(* Logix 5000 project; controller cal1632 1756-L62 rev 16.20; software revision 16.05; part 54 of 57 *)
(* tags used below, declared in another part *)
   FAULT : BOOL;
   p01_param_tension_deviation : REAL;
   p01r09_pb_global_reset : BOOL;
   p01r13_state : DINT;
   p25_ao_selected_speed : REAL;
   p29_ai_wa_rpm : REAL;
   p29_ai_wb_rpm : REAL;
   p29_ai_wdr_dia_in : REAL;
   p29_ai_wdr_lc : REAL;
   p29_di_wb_brake : BOOL;
   p29_di_wb_motor : BOOL;
   p29_di_wdr_a_core_size : BOOL;
   p29_di_wdr_a_reset_core : BOOL;
   p29_di_wdr_b_core_size : BOOL;
   p29_di_wdr_b_reset_core : BOOL;
   p29_di_wdr_index_fwd : BOOL;
   p29_param_wa_gear_ratio : REAL;
   p29_param_wb_gear_ratio : REAL;
   p29_wdb_status_word : INT;
   p29_wdb_vfd : ABB_PROTOCOL_VFD;
   p29r02_tension_dev_max : REAL;
   p29r02_tension_dev_min : REAL;
   p29r09_ten_ave_len : DINT;
   p29r09_ten_len : DINT;
   p29r09_ten_pos : DINT;
   p29r09_torque_mode : BOOL;
   p29r09_trq_ave_len : DINT;
   p29r09_trq_len : DINT;
   p29r09_trq_pos : DINT;
   p29r10_pid_psn : PID;
   p29r11_pid_psn : PID;
   p29r15_request_run : BOOL;
   p29r15_state : DINT;
   p29r16 : routine;
   p29r16_request_run : BOOL;
   p29r16_state : DINT;
   p29r16_timer_fault : TIMER[10];
   p29r16_timer_warning : TIMER[4];
   p29r17 : routine;
   p29r17_ave_control : CONTROL;
   p29r17_diameter_clac_active : BOOL;
   p29r17_selected_core_diameter : REAL;
   p29r17_stack_ctrl : CONTROL;
   p29r17_timer : TIMER[5];
   p29r17_timer_fault : TIMER[4];
   p29r17_timer_warning : TIMER[4];
   p29r17_winder_a_actual_diam_inch : REAL;
   p29r17_winder_a_avg_diam_inch : REAL;
   p29r17_winder_a_calc_diam_inch : REAL;
   p29r17_winder_a_diam_avg_stack : REAL[1000];
   p29r17_winder_a_selected_diam_inch : REAL;
   p29r17_winder_a_unload : REAL;
   p29r18 : routine;
   p29r18_ave_control : CONTROL;
   p29r18_diameter_calc_active : BOOL;
   p29r18_min_tension : REAL;
   p29r18_selected_core_diameter : REAL;
   p29r18_stack_ctrl : CONTROL;
   p29r18_timer : TIMER[5];
   p29r18_timer_fault : TIMER[4];
   p29r18_timer_warning : TIMER[4];
   p29r18_winder_b_actual_diam_inch : REAL;
   p29r18_winder_b_avg_diam_inch : REAL;
   p29r18_winder_b_calc_diam_inch : REAL;
   p29r18_winder_b_diam_avg_stack : REAL[1000];
   p29r18_winder_b_selected_diam_inch : REAL;
   p29r18_winder_b_unload : REAL;
   p29r20_index_complete : BOOL;
(* P29_Winder, continued *)

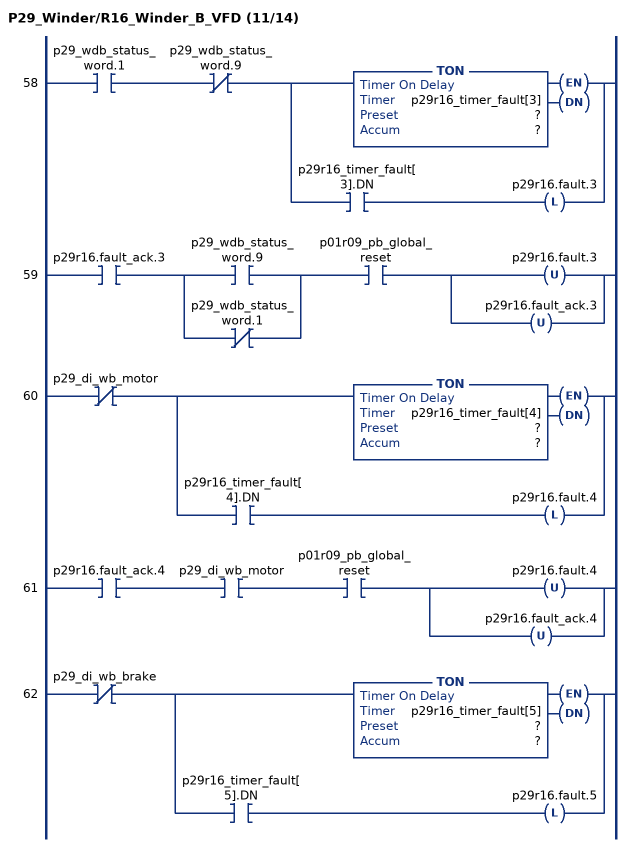
   [picture p1103: P29_Winder/R16_Winder_B_VFD rungs 58-62]
   58: XIC(p29_wdb_status_word.1)XIO(p29_wdb_status_word.9)[TON(p29r16_timer_fault[3],?,?) ,XIC(p29r16_timer_fault[3].DN) OTL(p29r16.fault.3) ];
   59: XIC(p29r16.fault_ack.3)[XIC(p29_wdb_status_word.9) ,XIO(p29_wdb_status_word.1) ]XIC(p01r09_pb_global_reset)[OTU(p29r16.fault.3) ,OTU(p29r16.fault_ack.3) ];
   60: XIO(p29_di_wb_motor)[TON(p29r16_timer_fault[4],?,?) ,XIC(p29r16_timer_fault[4].DN) OTL(p29r16.fault.4) ];
   61: XIC(p29r16.fault_ack.4)XIC(p29_di_wb_motor)XIC(p01r09_pb_global_reset)[OTU(p29r16.fault.4) ,OTU(p29r16.fault_ack.4) ];
   62: XIO(p29_di_wb_brake)[TON(p29r16_timer_fault[5],?,?) ,XIC(p29r16_timer_fault[5].DN) OTL(p29r16.fault.5) ];
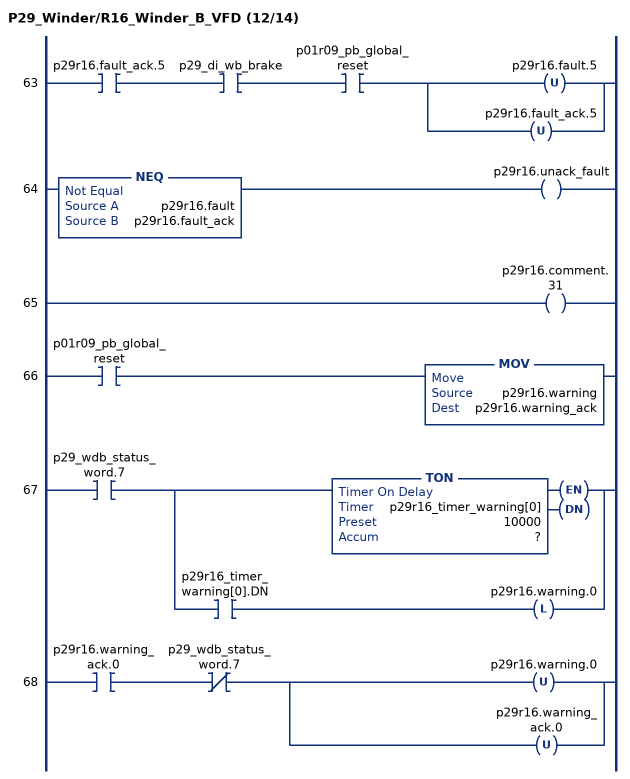
   63: XIC(p29r16.fault_ack.5)XIC(p29_di_wb_brake)XIC(p01r09_pb_global_reset)[OTU(p29r16.fault.5) ,OTU(p29r16.fault_ack.5) ];
   64: NEQ(p29r16.fault,p29r16.fault_ack)OTE(p29r16.unack_fault);
   65: OTE(p29r16.comment.31);
   66: XIC(p01r09_pb_global_reset)MOV(p29r16.warning,p29r16.warning_ack);
   67: XIC(p29_wdb_status_word.7)[TON(p29r16_timer_warning[0],?,?) ,XIC(p29r16_timer_warning[0].DN) OTL(p29r16.warning.0) ];
   68: XIC(p29r16.warning_ack.0)XIO(p29_wdb_status_word.7)[OTU(p29r16.warning.0) ,OTU(p29r16.warning_ack.0) ];
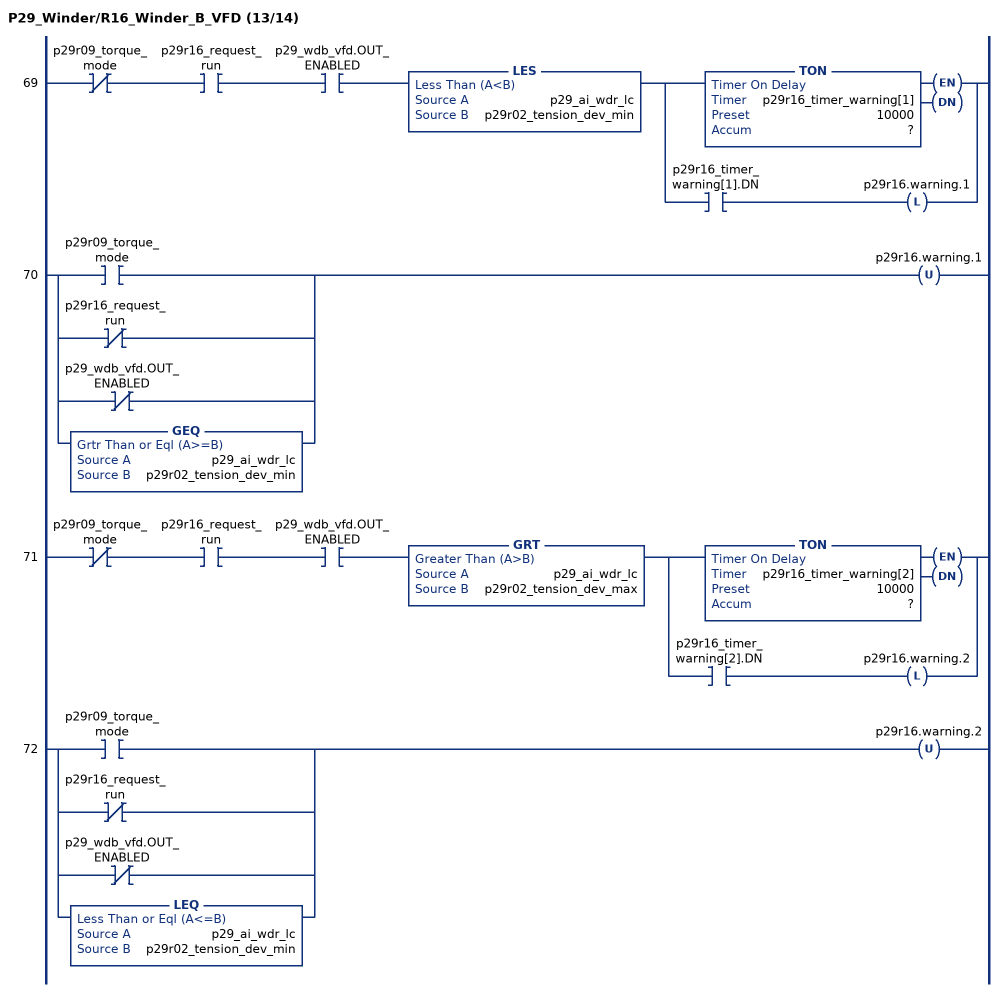
   69: XIO(p29r09_torque_mode)XIC(p29r16_request_run)XIC(p29_wdb_vfd.OUT_ENABLED)LES(p29_ai_wdr_lc,p29r02_tension_dev_min)[TON(p29r16_timer_warning[1],?,?) ,XIC(p29r16_timer_warning[1].DN) OTL(p29r16.warning.1) ];
   70: [XIC(p29r09_torque_mode) ,XIO(p29r16_request_run) ,XIO(p29_wdb_vfd.OUT_ENABLED) ,GEQ(p29_ai_wdr_lc,p29r02_tension_dev_min) ]OTU(p29r16.warning.1);
   71: XIO(p29r09_torque_mode)XIC(p29r16_request_run)XIC(p29_wdb_vfd.OUT_ENABLED)GRT(p29_ai_wdr_lc,p29r02_tension_dev_max)[TON(p29r16_timer_warning[2],?,?) ,XIC(p29r16_timer_warning[2].DN) OTL(p29r16.warning.2) ];
   72: [XIC(p29r09_torque_mode) ,XIO(p29r16_request_run) ,XIO(p29_wdb_vfd.OUT_ENABLED) ,LEQ(p29_ai_wdr_lc,p29r02_tension_dev_min) ]OTU(p29r16.warning.2);
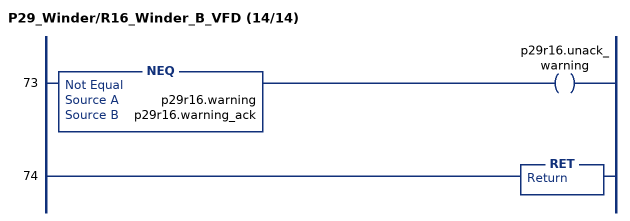
   73: NEQ(p29r16.warning,p29r16.warning_ack)OTE(p29r16.unack_warning);
   74: RET();
END_ROUTINE

ROUTINE R17_Winder_A_diameter_calc   (* ladder *)
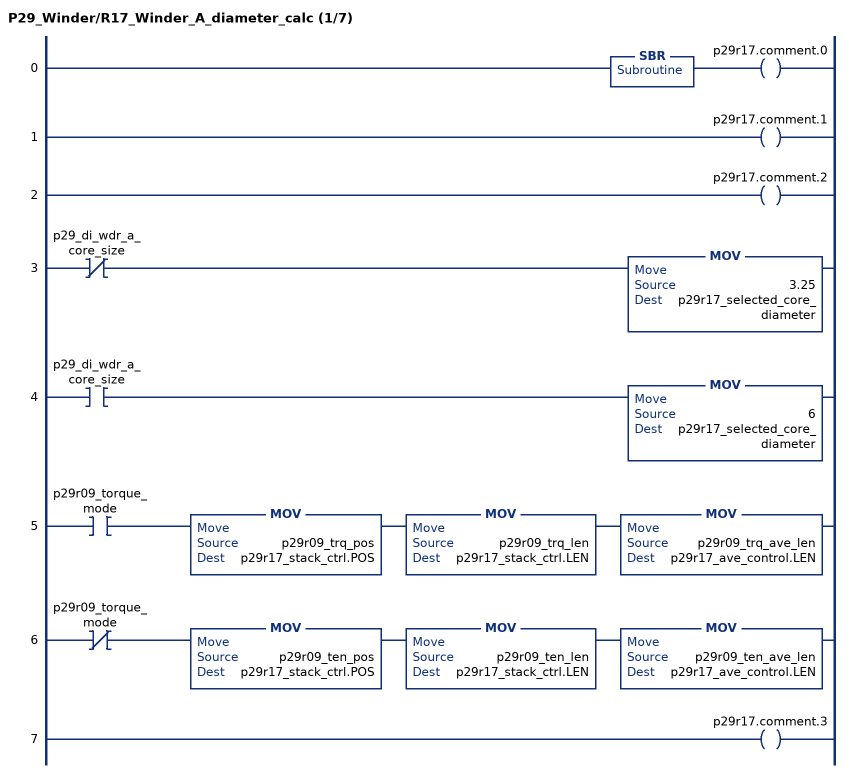
   0: SBR()OTE(p29r17.comment.0);
   1: OTE(p29r17.comment.1);
   2: OTE(p29r17.comment.2);
   3: XIO(p29_di_wdr_a_core_size)MOV(3.25,p29r17_selected_core_diameter);
   4: XIC(p29_di_wdr_a_core_size)MOV(6,p29r17_selected_core_diameter);
   5: XIC(p29r09_torque_mode)MOV(p29r09_trq_pos,p29r17_stack_ctrl.POS)MOV(p29r09_trq_len,p29r17_stack_ctrl.LEN)MOV(p29r09_trq_ave_len,p29r17_ave_control.LEN);
   6: XIO(p29r09_torque_mode)MOV(p29r09_ten_pos,p29r17_stack_ctrl.POS)MOV(p29r09_ten_len,p29r17_stack_ctrl.LEN)MOV(p29r09_ten_ave_len,p29r17_ave_control.LEN);
   7: OTE(p29r17.comment.3);
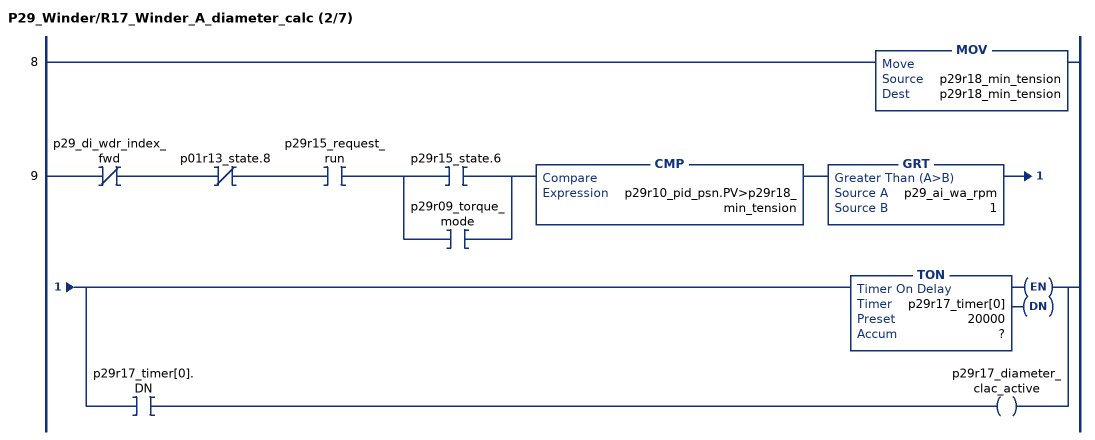
   8: MOV(p29r18_min_tension,p29r18_min_tension);
   9: XIO(p29_di_wdr_index_fwd)XIO(p01r13_state.8)XIC(p29r15_request_run)[XIC(p29r15_state.6) ,XIC(p29r09_torque_mode) ]CMP(p29r10_pid_psn.PV>p29r18_min_tension)GRT(p29_ai_wa_rpm,1)[TON(p29r17_timer[0],?,?) ,XIC(p29r17_timer[0].DN) OTE(p29r17_diameter_clac_active) ];
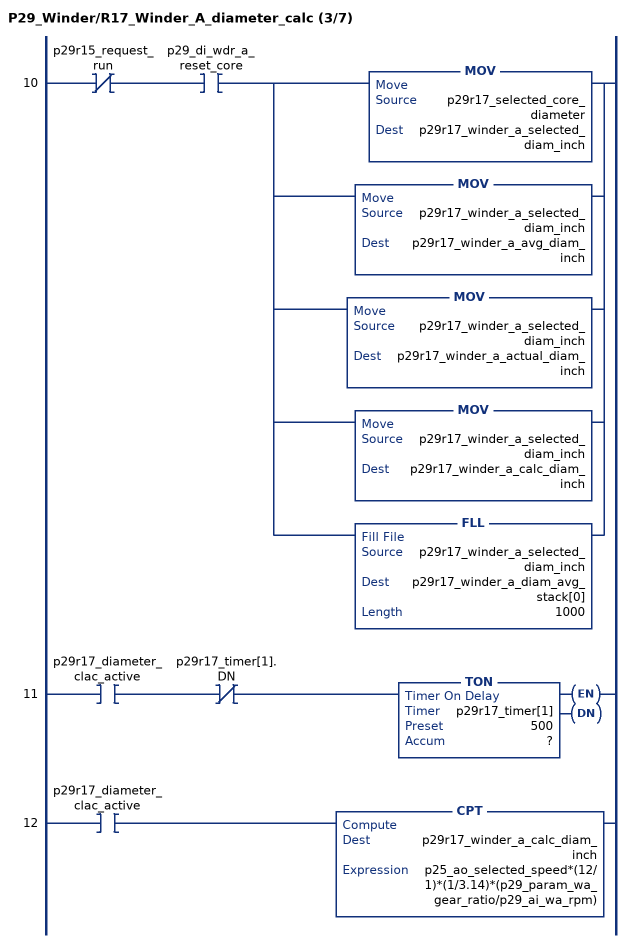
   10: XIO(p29r15_request_run)XIC(p29_di_wdr_a_reset_core)[MOV(p29r17_selected_core_diameter,p29r17_winder_a_selected_diam_inch) ,MOV(p29r17_winder_a_selected_diam_inch,p29r17_winder_a_avg_diam_inch) ,MOV(p29r17_winder_a_selected_diam_inch,p29r17_winder_a_actual_diam_inch) ,MOV(p29r17_winder_a_selected_diam_inch,p29r17_winder_a_calc_diam_inch) ,FLL(p29r17_winder_a_selected_diam_inch,p29r17_winder_a_diam_avg_stack[0],1000) ];
   11: XIC(p29r17_diameter_clac_active)XIO(p29r17_timer[1].DN)TON(p29r17_timer[1],?,?);
   12: XIC(p29r17_diameter_clac_active)CPT(p29r17_winder_a_calc_diam_inch,p25_ao_selected_speed*(12/1)*(1/3.14)*(p29_param_wa_gear_ratio/p29_ai_wa_rpm));
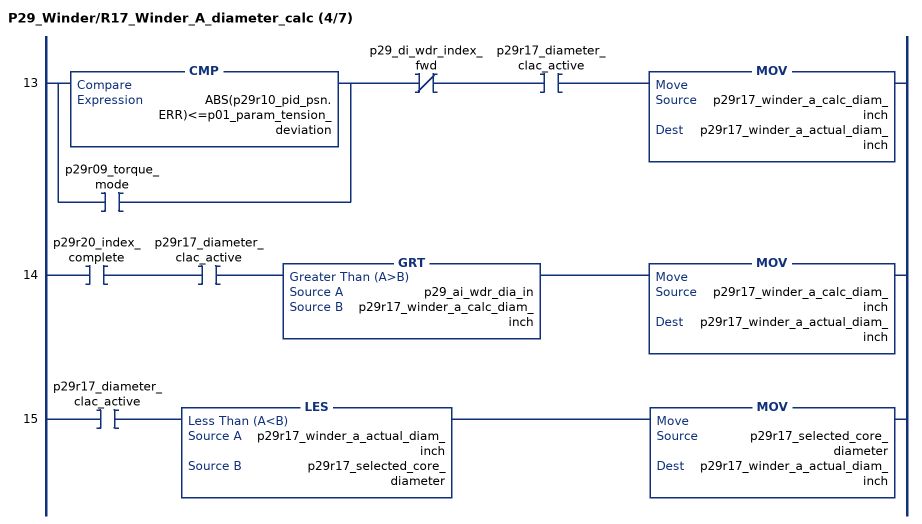
   13: [CMP(ABS(p29r10_pid_psn.ERR)<=p01_param_tension_deviation) ,XIC(p29r09_torque_mode) ]XIO(p29_di_wdr_index_fwd)XIC(p29r17_diameter_clac_active)MOV(p29r17_winder_a_calc_diam_inch,p29r17_winder_a_actual_diam_inch);
   14: XIC(p29r20_index_complete)XIC(p29r17_diameter_clac_active)GRT(p29_ai_wdr_dia_in,p29r17_winder_a_calc_diam_inch)MOV(p29r17_winder_a_calc_diam_inch,p29r17_winder_a_actual_diam_inch);
   15: XIC(p29r17_diameter_clac_active)LES(p29r17_winder_a_actual_diam_inch,p29r17_selected_core_diameter)MOV(p29r17_selected_core_diameter,p29r17_winder_a_actual_diam_inch);
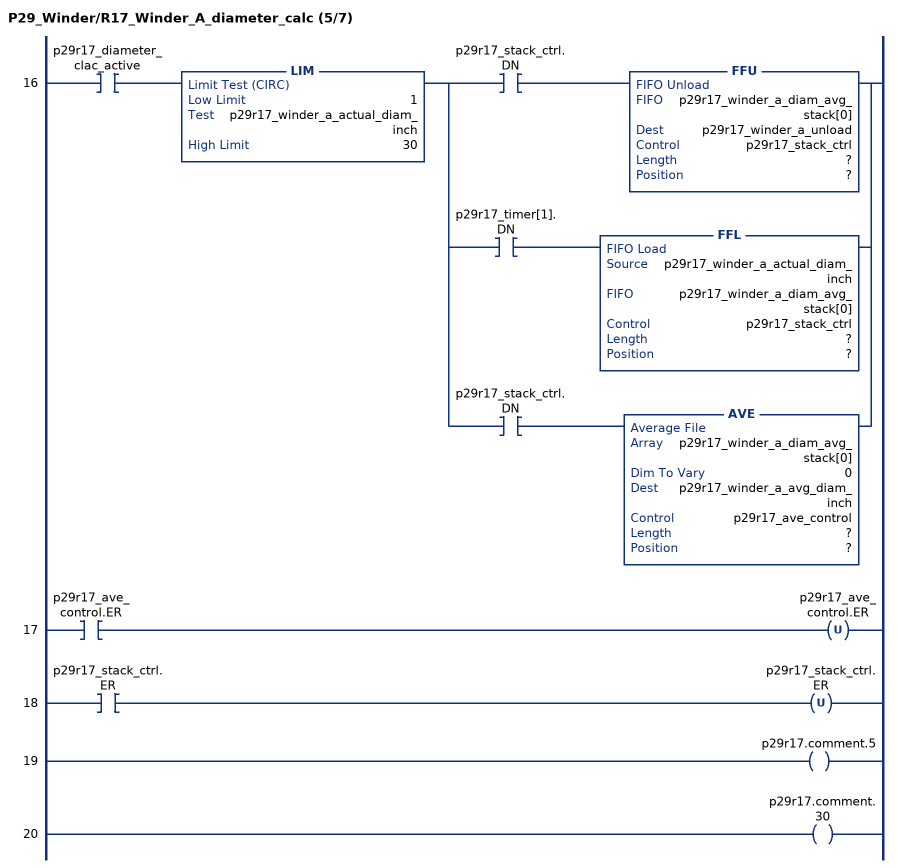
   16: XIC(p29r17_diameter_clac_active)LIM(1,p29r17_winder_a_actual_diam_inch,30)[XIC(p29r17_stack_ctrl.DN) FFU(p29r17_winder_a_diam_avg_stack[0],p29r17_winder_a_unload,p29r17_stack_ctrl,?,?) ,XIC(p29r17_timer[1].DN) FFL(p29r17_winder_a_actual_diam_inch,p29r17_winder_a_diam_avg_stack[0],p29r17_stack_ctrl,?,?) ,XIC(p29r17_stack_ctrl.DN) AVE(p29r17_winder_a_diam_avg_stack[0],0,p29r17_winder_a_avg_diam_inch,p29r17_ave_control,?,?) ];
   17: XIC(p29r17_ave_control.ER)OTU(p29r17_ave_control.ER);
   18: XIC(p29r17_stack_ctrl.ER)OTU(p29r17_stack_ctrl.ER);
   19: OTE(p29r17.comment.5);
   20: OTE(p29r17.comment.30);
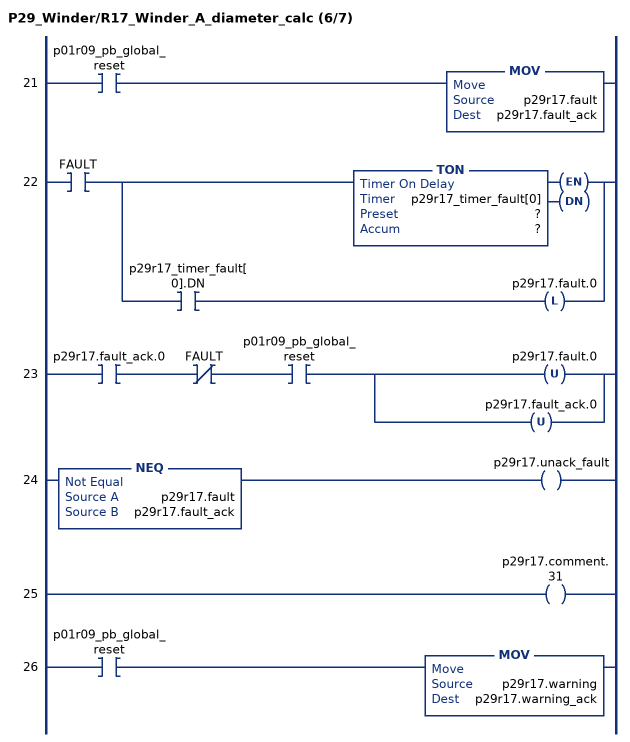
   21: XIC(p01r09_pb_global_reset)MOV(p29r17.fault,p29r17.fault_ack);
   22: XIC(FAULT)[TON(p29r17_timer_fault[0],?,?) ,XIC(p29r17_timer_fault[0].DN) OTL(p29r17.fault.0) ];
   23: XIC(p29r17.fault_ack.0)XIO(FAULT)XIC(p01r09_pb_global_reset)[OTU(p29r17.fault.0) ,OTU(p29r17.fault_ack.0) ];
   24: NEQ(p29r17.fault,p29r17.fault_ack)OTE(p29r17.unack_fault);
   25: OTE(p29r17.comment.31);
   26: XIC(p01r09_pb_global_reset)MOV(p29r17.warning,p29r17.warning_ack);
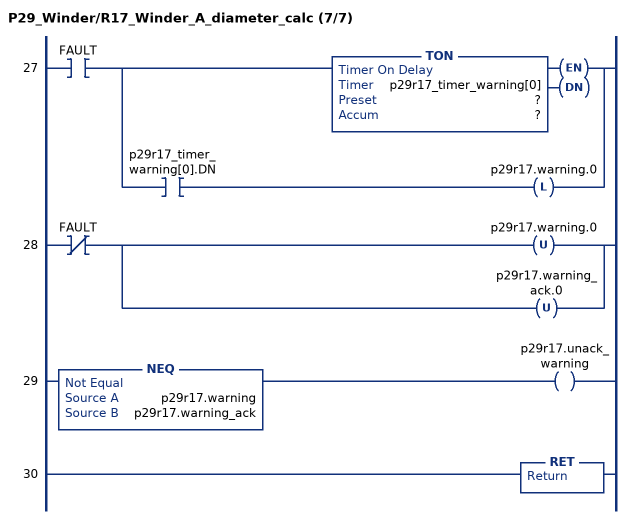
   27: XIC(FAULT)[TON(p29r17_timer_warning[0],?,?) ,XIC(p29r17_timer_warning[0].DN) OTL(p29r17.warning.0) ];
   28: XIO(FAULT)[OTU(p29r17.warning.0) ,OTU(p29r17.warning_ack.0) ];
   29: NEQ(p29r17.warning,p29r17.warning_ack)OTE(p29r17.unack_warning);
   30: RET();
END_ROUTINE

ROUTINE R18_Winder_B_diameter_calc   (* ladder *)
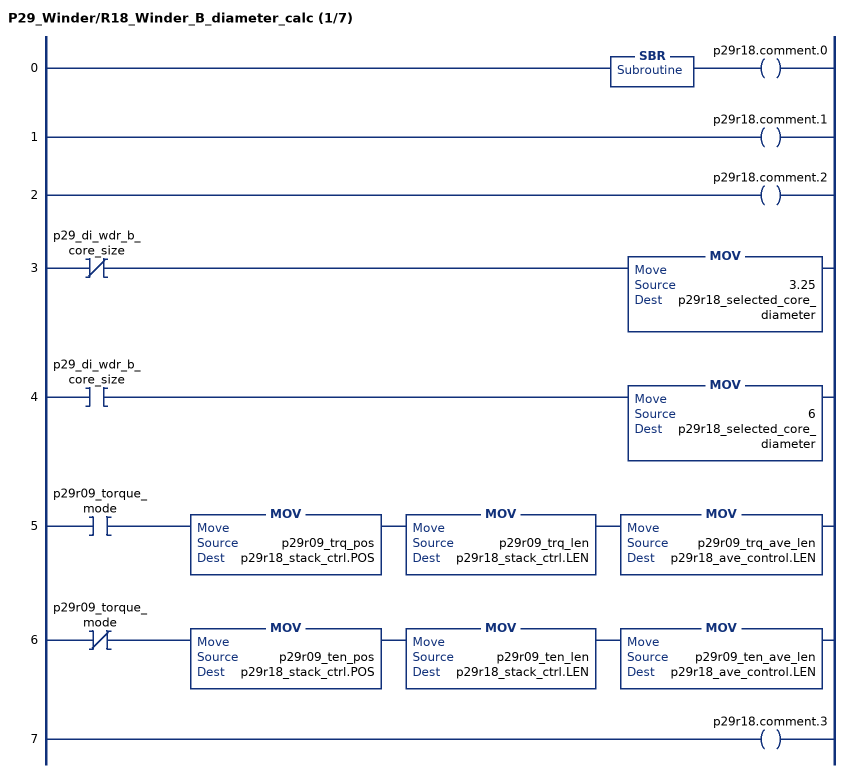
   0: SBR()OTE(p29r18.comment.0);
   1: OTE(p29r18.comment.1);
   2: OTE(p29r18.comment.2);
   3: XIO(p29_di_wdr_b_core_size)MOV(3.25,p29r18_selected_core_diameter);
   4: XIC(p29_di_wdr_b_core_size)MOV(6,p29r18_selected_core_diameter);
   5: XIC(p29r09_torque_mode)MOV(p29r09_trq_pos,p29r18_stack_ctrl.POS)MOV(p29r09_trq_len,p29r18_stack_ctrl.LEN)MOV(p29r09_trq_ave_len,p29r18_ave_control.LEN);
   6: XIO(p29r09_torque_mode)MOV(p29r09_ten_pos,p29r18_stack_ctrl.POS)MOV(p29r09_ten_len,p29r18_stack_ctrl.LEN)MOV(p29r09_ten_ave_len,p29r18_ave_control.LEN);
   7: OTE(p29r18.comment.3);
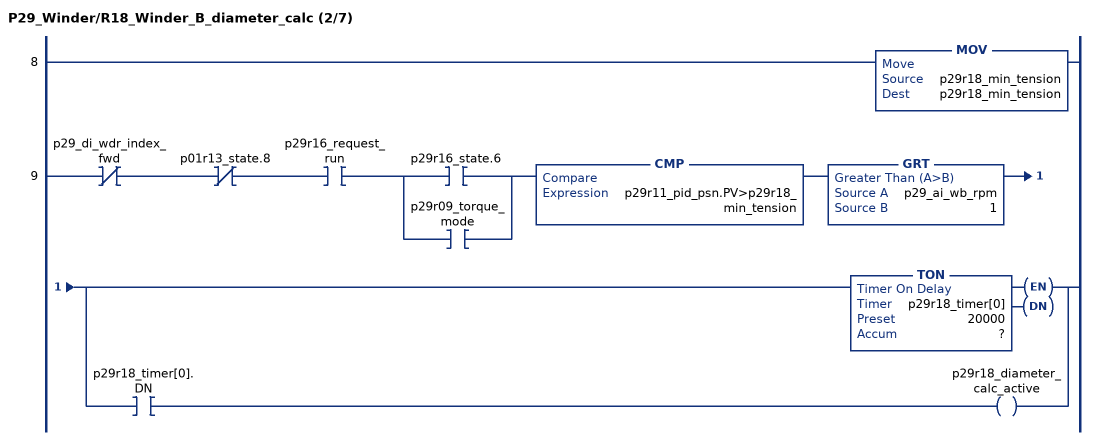
   8: MOV(p29r18_min_tension,p29r18_min_tension);
   9: XIO(p29_di_wdr_index_fwd)XIO(p01r13_state.8)XIC(p29r16_request_run)[XIC(p29r16_state.6) ,XIC(p29r09_torque_mode) ]CMP(p29r11_pid_psn.PV>p29r18_min_tension)GRT(p29_ai_wb_rpm,1)[TON(p29r18_timer[0],?,?) ,XIC(p29r18_timer[0].DN) OTE(p29r18_diameter_calc_active) ];
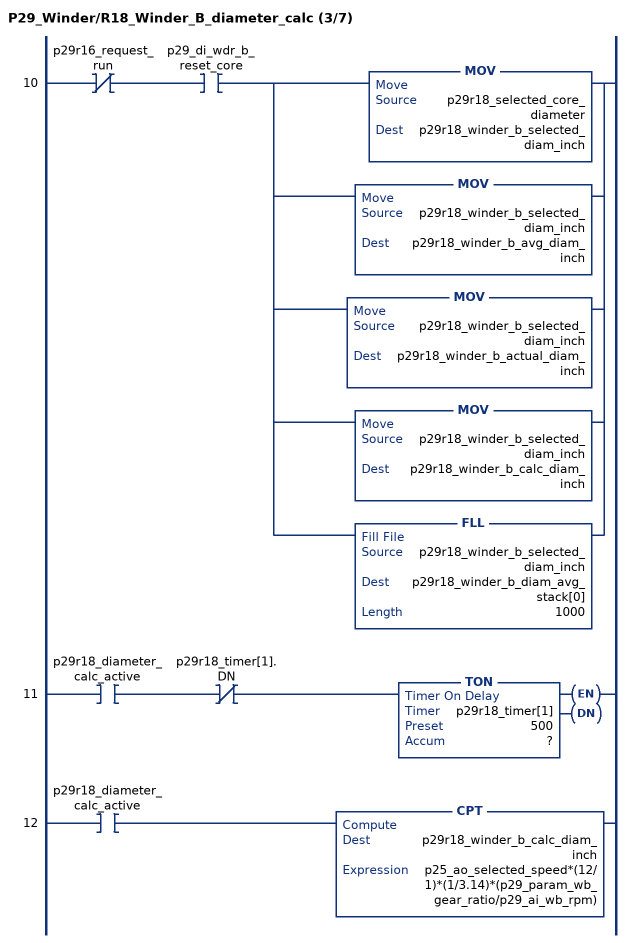
   10: XIO(p29r16_request_run)XIC(p29_di_wdr_b_reset_core)[MOV(p29r18_selected_core_diameter,p29r18_winder_b_selected_diam_inch) ,MOV(p29r18_winder_b_selected_diam_inch,p29r18_winder_b_avg_diam_inch) ,MOV(p29r18_winder_b_selected_diam_inch,p29r18_winder_b_actual_diam_inch) ,MOV(p29r18_winder_b_selected_diam_inch,p29r18_winder_b_calc_diam_inch) ,FLL(p29r18_winder_b_selected_diam_inch,p29r18_winder_b_diam_avg_stack[0],1000) ];
   11: XIC(p29r18_diameter_calc_active)XIO(p29r18_timer[1].DN)TON(p29r18_timer[1],?,?);
   12: XIC(p29r18_diameter_calc_active)CPT(p29r18_winder_b_calc_diam_inch,p25_ao_selected_speed*(12/1)*(1/3.14)*(p29_param_wb_gear_ratio/p29_ai_wb_rpm));
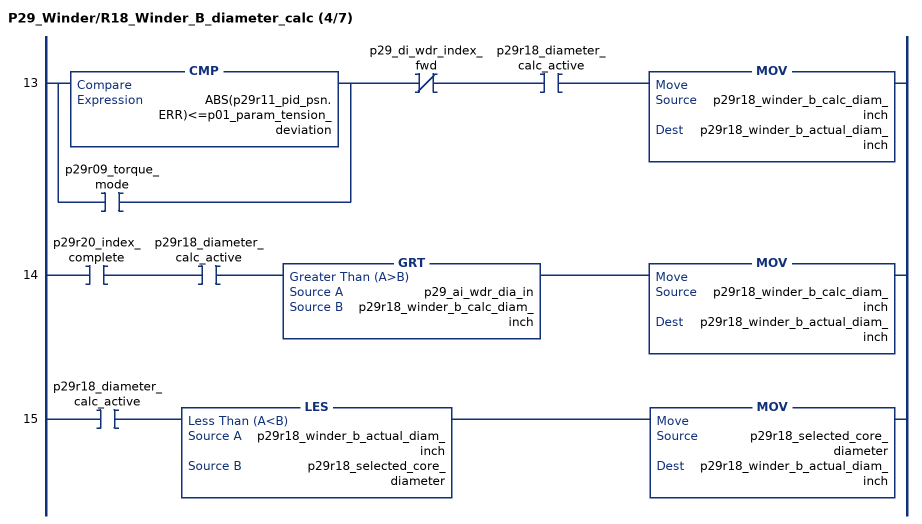
   13: [CMP(ABS(p29r11_pid_psn.ERR)<=p01_param_tension_deviation) ,XIC(p29r09_torque_mode) ]XIO(p29_di_wdr_index_fwd)XIC(p29r18_diameter_calc_active)MOV(p29r18_winder_b_calc_diam_inch,p29r18_winder_b_actual_diam_inch);
   14: XIC(p29r20_index_complete)XIC(p29r18_diameter_calc_active)GRT(p29_ai_wdr_dia_in,p29r18_winder_b_calc_diam_inch)MOV(p29r18_winder_b_calc_diam_inch,p29r18_winder_b_actual_diam_inch);
   15: XIC(p29r18_diameter_calc_active)LES(p29r18_winder_b_actual_diam_inch,p29r18_selected_core_diameter)MOV(p29r18_selected_core_diameter,p29r18_winder_b_actual_diam_inch);
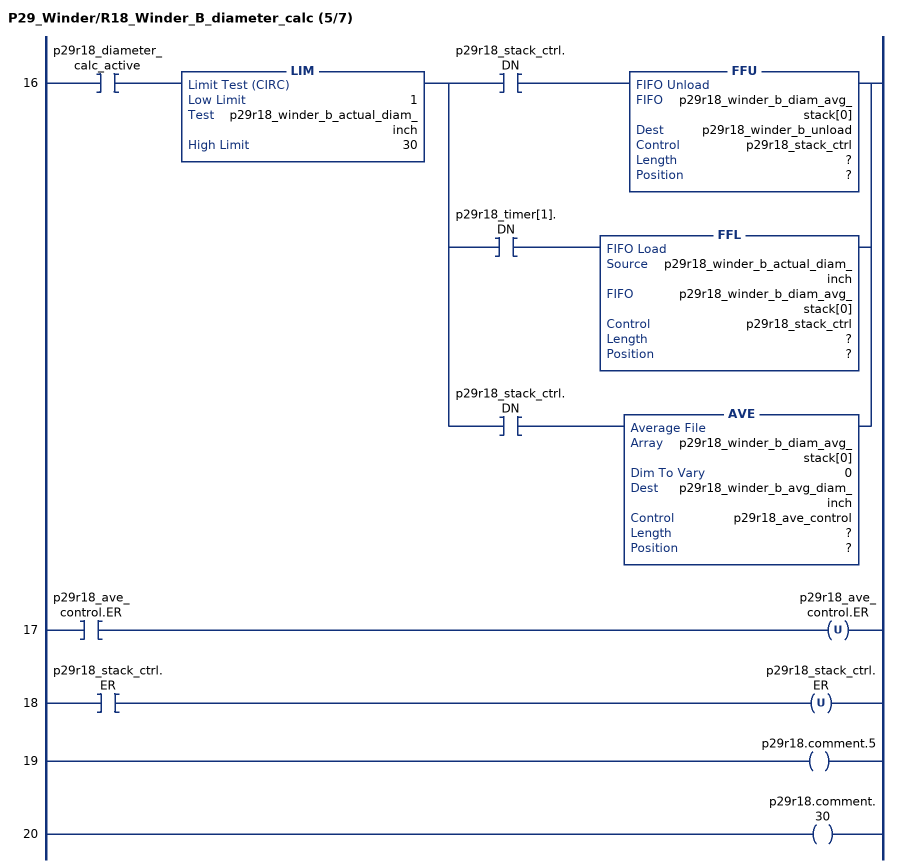
   16: XIC(p29r18_diameter_calc_active)LIM(1,p29r18_winder_b_actual_diam_inch,30)[XIC(p29r18_stack_ctrl.DN) FFU(p29r18_winder_b_diam_avg_stack[0],p29r18_winder_b_unload,p29r18_stack_ctrl,?,?) ,XIC(p29r18_timer[1].DN) FFL(p29r18_winder_b_actual_diam_inch,p29r18_winder_b_diam_avg_stack[0],p29r18_stack_ctrl,?,?) ,XIC(p29r18_stack_ctrl.DN) AVE(p29r18_winder_b_diam_avg_stack[0],0,p29r18_winder_b_avg_diam_inch,p29r18_ave_control,?,?) ];
   17: XIC(p29r18_ave_control.ER)OTU(p29r18_ave_control.ER);
   18: XIC(p29r18_stack_ctrl.ER)OTU(p29r18_stack_ctrl.ER);
   19: OTE(p29r18.comment.5);
   20: OTE(p29r18.comment.30);
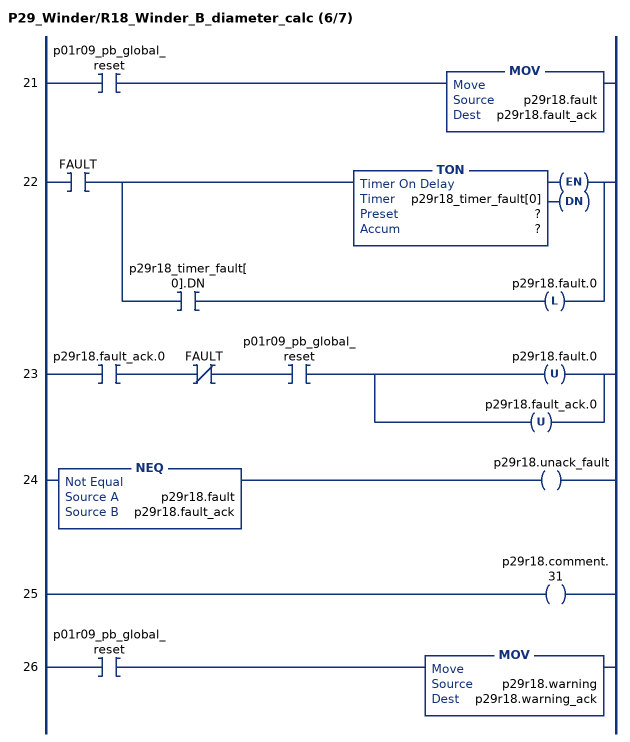
   21: XIC(p01r09_pb_global_reset)MOV(p29r18.fault,p29r18.fault_ack);
   22: XIC(FAULT)[TON(p29r18_timer_fault[0],?,?) ,XIC(p29r18_timer_fault[0].DN) OTL(p29r18.fault.0) ];
   23: XIC(p29r18.fault_ack.0)XIO(FAULT)XIC(p01r09_pb_global_reset)[OTU(p29r18.fault.0) ,OTU(p29r18.fault_ack.0) ];
   24: NEQ(p29r18.fault,p29r18.fault_ack)OTE(p29r18.unack_fault);
   25: OTE(p29r18.comment.31);
   26: XIC(p01r09_pb_global_reset)MOV(p29r18.warning,p29r18.warning_ack);
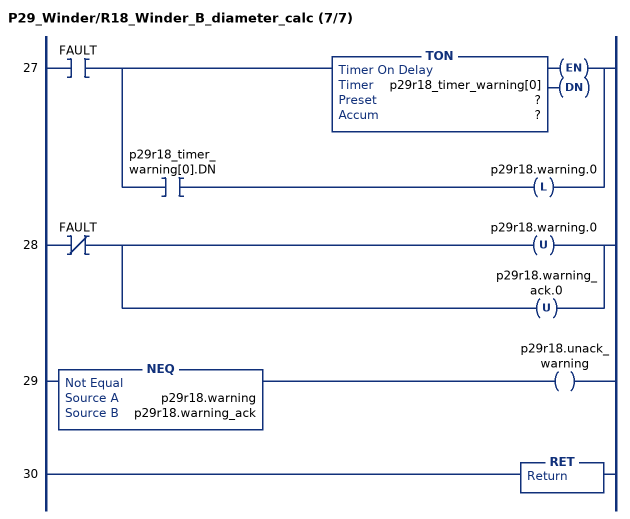
   27: XIC(FAULT)[TON(p29r18_timer_warning[0],?,?) ,XIC(p29r18_timer_warning[0].DN) OTL(p29r18.warning.0) ];
   28: XIO(FAULT)[OTU(p29r18.warning.0) ,OTU(p29r18.warning_ack.0) ];
   29: NEQ(p29r18.warning,p29r18.warning_ack)OTE(p29r18.unack_warning);
   30: RET();
END_ROUTINE
